Staubli VAL3: PerforatiAction.pgx

public program PerforatiAction(num x_nGasDelay (dimensions=1), num x_nFollowDelay (dimensions=1))
begin

  //穿孔动作
  call KeyDigtalIO(true,true,true,x_nGasDelay,x_nFollowDelay)

end
